// TIA Portal V16 export
// export: Created 2024-09-05T17:40:14.9004308Z, ExportSetting WithDefaults, DisplayName Totally Integrated Automation Portal, DisplayVersion V16 Update 6, DisplayName TIA Portal Version Control Interface, DisplayVersion V16 Update 2, DisplayName TIA Portal Openness, DisplayVersion V16 Update 6, DisplayName STEP 7 Professional, DisplayVersion V16 Update 6, DisplayName STEP 7 Safety, DisplayVersion V16, DisplayName WinCC Advanced, DisplayVersion V16 Update 6
TYPE "UDT_HMI"
// stored: IsFailsafeCompliant false
   STRUCT
      ScreenData : Array[1..5] of Word;
      UserNumber : UInt;
      ActualScreenNumber : UInt;
      RequiredScreenNumber : UInt;
      FunctionKeys : Array[1..8] of Bool;
   END_STRUCT;
END_TYPE
